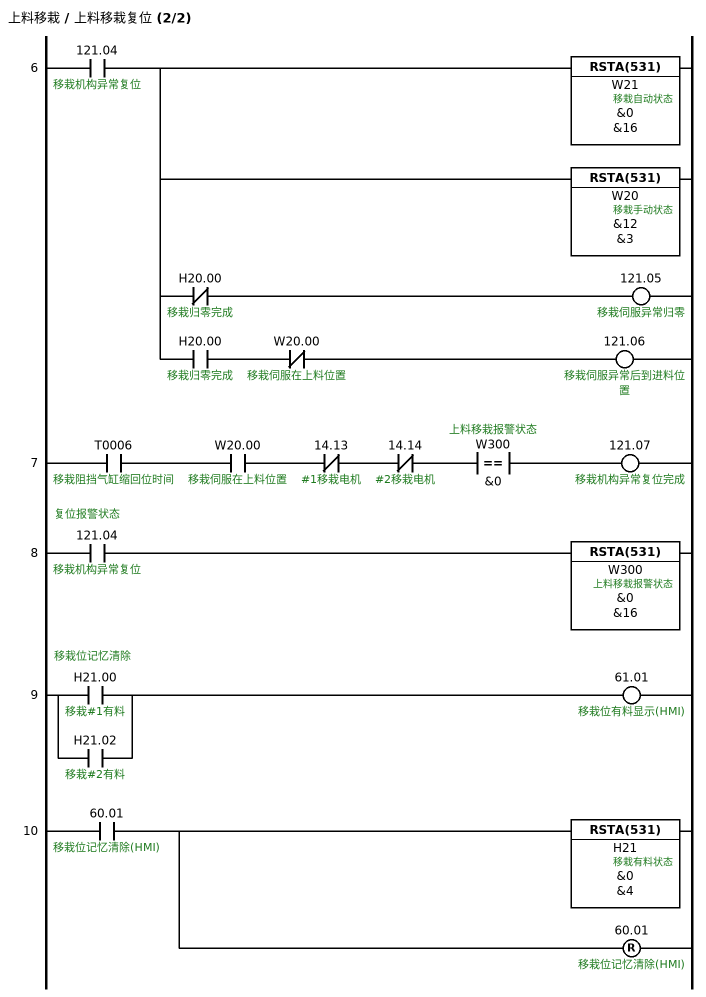
; [picture p113: 上料移栽 / 上料移栽复位, rungs 6-10]
; rung 6
LD 121.04  ; 移栽机构异常复位
OUT TR0
RSTA(531) W21 &0 &16  ; 移栽自动状态
RSTA(531) W20 &12 &3  ; 移栽手动状态
ANDNOT H20.00  ; 移栽归零完成
OUT 121.05  ; 移栽伺服异常归零
LD TR0
AND H20.00  ; 移栽归零完成
ANDNOT W20.00  ; 移栽伺服在上料位置
OUT 121.06  ; 移栽伺服异常后到进料位置
; rung 7
LD T0006  ; 移栽阻挡气缸缩回位时间
AND W20.00  ; 移栽伺服在上料位置
ANDNOT 14.13  ; #1移栽电机
ANDNOT 14.14  ; #2移栽电机
AND=(300) W300 &0  ; 上料移栽报警状态
OUT 121.07  ; 移栽机构异常复位完成
; rung 8: 复位报警状态
LD 121.04  ; 移栽机构异常复位
RSTA(531) W300 &0 &16  ; 上料移栽报警状态
; rung 9: 移栽位记忆清除
LD H21.00  ; 移栽#1有料
OR H21.02  ; 移栽#2有料
OUT 61.01  ; 移栽位有料显示(HMI)
; rung 10
LD 60.01  ; 移栽位记忆清除(HMI)
RSTA(531) H21 &0 &4  ; 移栽有料状态
RSET 60.01  ; 移栽位记忆清除(HMI)

### Section END
; rung 0
END(001)

## Program 左机械手 (cyclic task 4)

### Section 左机械手手动

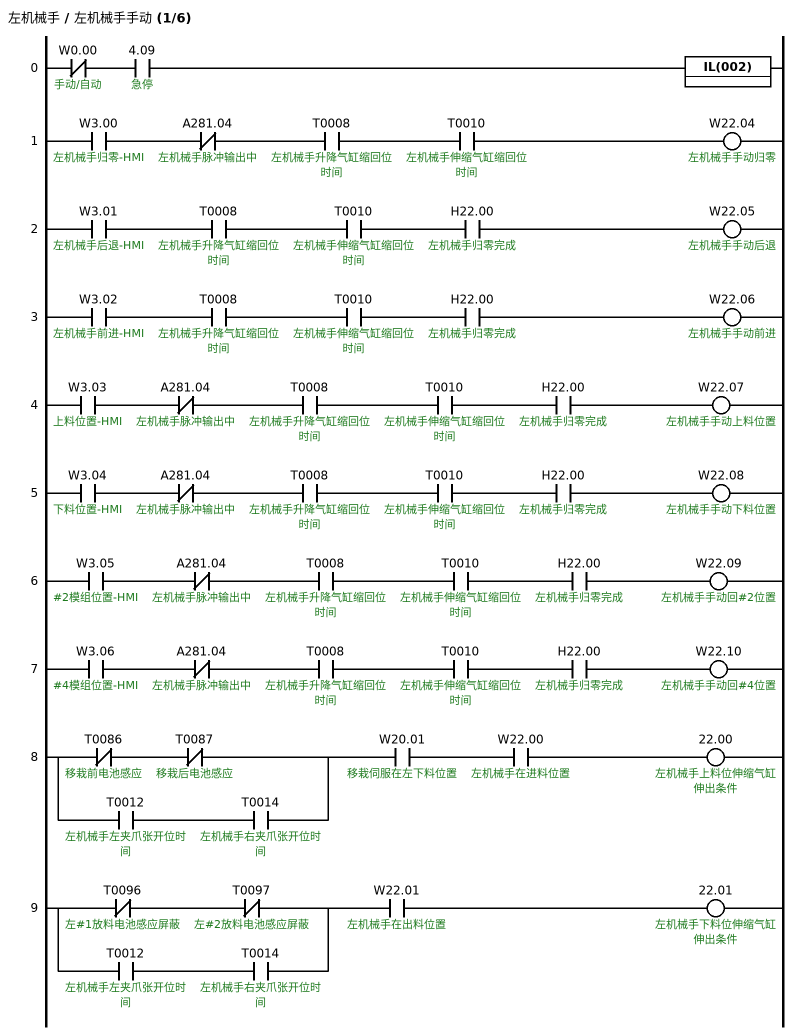
; rung 0
LDNOT W0.00  ; 手动/自动
AND 4.09  ; 急停
IL(002)
; rung 1
LD W3.00  ; 左机械手归零-HMI
ANDNOT A281.04  ; 左机械手脉冲输出中
AND T0008  ; 左机械手升降气缸缩回位时间
AND T0010  ; 左机械手伸缩气缸缩回位时间
OUT W22.04  ; 左机械手手动归零
; rung 2
LD W3.01  ; 左机械手后退-HMI
AND T0008  ; 左机械手升降气缸缩回位时间
AND T0010  ; 左机械手伸缩气缸缩回位时间
AND H22.00  ; 左机械手归零完成
OUT W22.05  ; 左机械手手动后退
; rung 3
LD W3.02  ; 左机械手前进-HMI
AND T0008  ; 左机械手升降气缸缩回位时间
AND T0010  ; 左机械手伸缩气缸缩回位时间
AND H22.00  ; 左机械手归零完成
OUT W22.06  ; 左机械手手动前进
; rung 4
LD W3.03  ; 上料位置-HMI
ANDNOT A281.04  ; 左机械手脉冲输出中
AND T0008  ; 左机械手升降气缸缩回位时间
AND T0010  ; 左机械手伸缩气缸缩回位时间
AND H22.00  ; 左机械手归零完成
OUT W22.07  ; 左机械手手动上料位置
; rung 5
LD W3.04  ; 下料位置-HMI
ANDNOT A281.04  ; 左机械手脉冲输出中
AND T0008  ; 左机械手升降气缸缩回位时间
AND T0010  ; 左机械手伸缩气缸缩回位时间
AND H22.00  ; 左机械手归零完成
OUT W22.08  ; 左机械手手动下料位置
; rung 6
LD W3.05  ; #2模组位置-HMI
ANDNOT A281.04  ; 左机械手脉冲输出中
AND T0008  ; 左机械手升降气缸缩回位时间
AND T0010  ; 左机械手伸缩气缸缩回位时间
AND H22.00  ; 左机械手归零完成
OUT W22.09  ; 左机械手手动回#2位置
; rung 7
LD W3.06  ; #4模组位置-HMI
ANDNOT A281.04  ; 左机械手脉冲输出中
AND T0008  ; 左机械手升降气缸缩回位时间
AND T0010  ; 左机械手伸缩气缸缩回位时间
AND H22.00  ; 左机械手归零完成
OUT W22.10  ; 左机械手手动回#4位置
; rung 8
LDNOT T0086  ; 移栽前电池感应
ANDNOT T0087  ; 移栽后电池感应
LD T0012  ; 左机械手左夹爪张开位时间
AND T0014  ; 左机械手右夹爪张开位时间
ORLD
AND W20.01  ; 移栽伺服在左下料位置
AND W22.00  ; 左机械手在进料位置
OUT 22.00  ; 左机械手上料位伸缩气缸伸出条件
; rung 9
LDNOT T0096  ; 左#1放料电池感应屏蔽
ANDNOT T0097  ; 左#2放料电池感应屏蔽
LD T0012  ; 左机械手左夹爪张开位时间
AND T0014  ; 左机械手右夹爪张开位时间
ORLD
AND W22.01  ; 左机械手在出料位置
OUT 22.01  ; 左机械手下料位伸缩气缸伸出条件

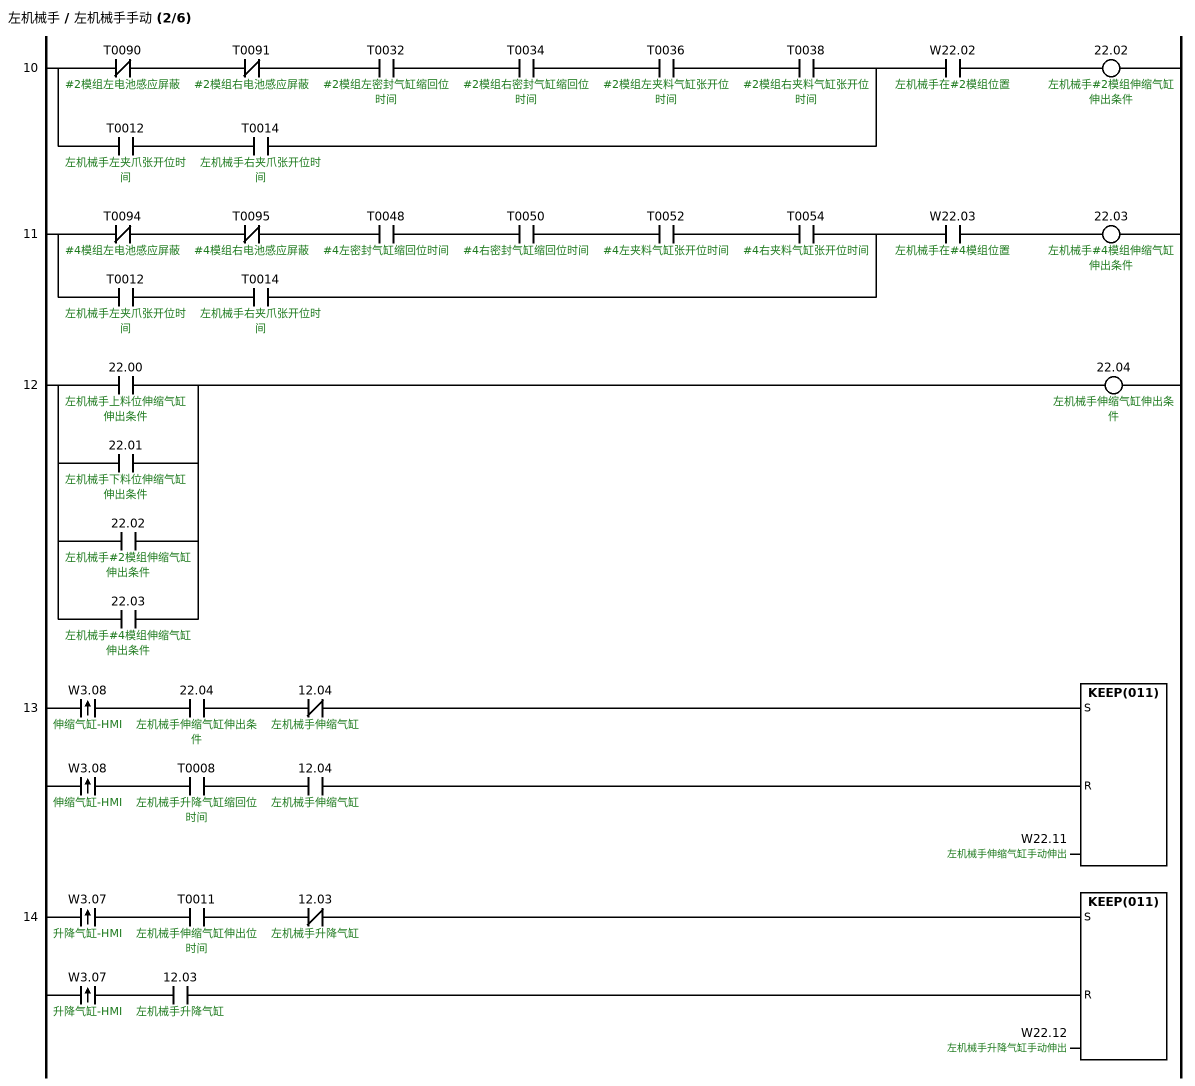
; rung 10
LDNOT T0090  ; #2模组左电池感应屏蔽
ANDNOT T0091  ; #2模组右电池感应屏蔽
AND T0032  ; #2模组左密封气缸缩回位时间
AND T0034  ; #2模组右密封气缸缩回位时间
AND T0036  ; #2模组左夹料气缸张开位时间
AND T0038  ; #2模组右夹料气缸张开位时间
LD T0012  ; 左机械手左夹爪张开位时间
AND T0014  ; 左机械手右夹爪张开位时间
ORLD
AND W22.02  ; 左机械手在#2模组位置
OUT 22.02  ; 左机械手#2模组伸缩气缸伸出条件
; rung 11
LDNOT T0094  ; #4模组左电池感应屏蔽
ANDNOT T0095  ; #4模组右电池感应屏蔽
AND T0048  ; #4左密封气缸缩回位时间
AND T0050  ; #4右密封气缸缩回位时间
AND T0052  ; #4左夹料气缸张开位时间
AND T0054  ; #4右夹料气缸张开位时间
LD T0012  ; 左机械手左夹爪张开位时间
AND T0014  ; 左机械手右夹爪张开位时间
ORLD
AND W22.03  ; 左机械手在#4模组位置
OUT 22.03  ; 左机械手#4模组伸缩气缸伸出条件
; rung 12
LD 22.00  ; 左机械手上料位伸缩气缸伸出条件
OR 22.01  ; 左机械手下料位伸缩气缸伸出条件
OR 22.02  ; 左机械手#2模组伸缩气缸伸出条件
OR 22.03  ; 左机械手#4模组伸缩气缸伸出条件
OUT 22.04  ; 左机械手伸缩气缸伸出条件
; rung 13
@LD W3.08  ; 伸缩气缸-HMI
AND 22.04  ; 左机械手伸缩气缸伸出条件
ANDNOT 12.04  ; 左机械手伸缩气缸
@LD W3.08  ; 伸缩气缸-HMI
AND T0008  ; 左机械手升降气缸缩回位时间
AND 12.04  ; 左机械手伸缩气缸
KEEP(011) W22.11  ; 左机械手伸缩气缸手动伸出
; rung 14
@LD W3.07  ; 升降气缸-HMI
AND T0011  ; 左机械手伸缩气缸伸出位时间
ANDNOT 12.03  ; 左机械手升降气缸
@LD W3.07  ; 升降气缸-HMI
AND 12.03  ; 左机械手升降气缸
KEEP(011) W22.12  ; 左机械手升降气缸手动伸出

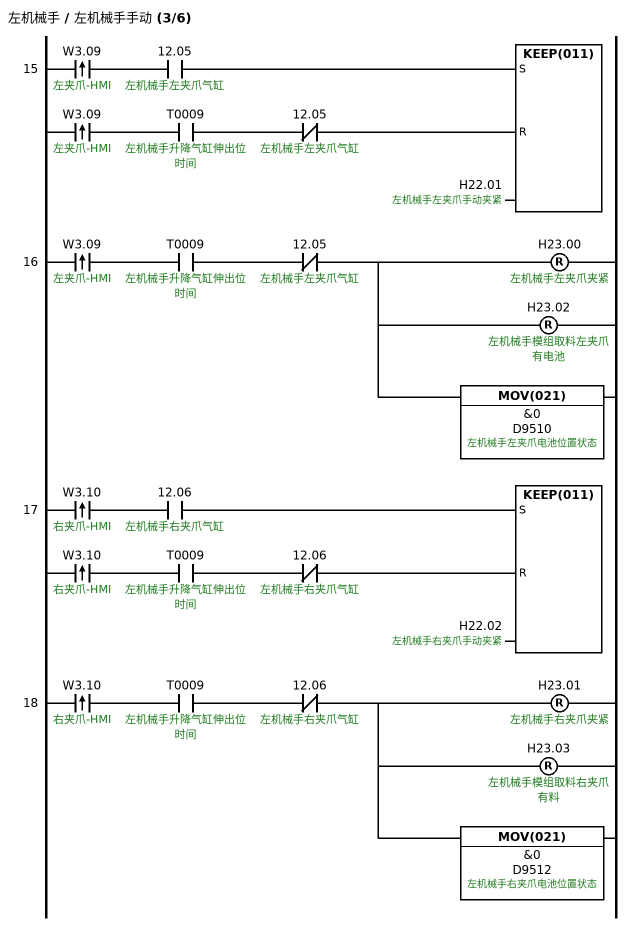
; rung 15
@LD W3.09  ; 左夹爪-HMI
AND 12.05  ; 左机械手左夹爪气缸
@LD W3.09  ; 左夹爪-HMI
AND T0009  ; 左机械手升降气缸伸出位时间
ANDNOT 12.05  ; 左机械手左夹爪气缸
KEEP(011) H22.01  ; 左机械手左夹爪手动夹紧
; rung 16
@LD W3.09  ; 左夹爪-HMI
AND T0009  ; 左机械手升降气缸伸出位时间
ANDNOT 12.05  ; 左机械手左夹爪气缸
RSET H23.00  ; 左机械手左夹爪夹紧
RSET H23.02  ; 左机械手模组取料左夹爪有电池
MOV(021) &0 D9510  ; 左机械手左夹爪电池位置状态
; rung 17
@LD W3.10  ; 右夹爪-HMI
AND 12.06  ; 左机械手右夹爪气缸
@LD W3.10  ; 右夹爪-HMI
AND T0009  ; 左机械手升降气缸伸出位时间
ANDNOT 12.06  ; 左机械手右夹爪气缸
KEEP(011) H22.02  ; 左机械手右夹爪手动夹紧
; rung 18
@LD W3.10  ; 右夹爪-HMI
AND T0009  ; 左机械手升降气缸伸出位时间
ANDNOT 12.06  ; 左机械手右夹爪气缸
RSET H23.01  ; 左机械手右夹爪夹紧
RSET H23.03  ; 左机械手模组取料右夹爪有料
MOV(021) &0 D9512  ; 左机械手右夹爪电池位置状态

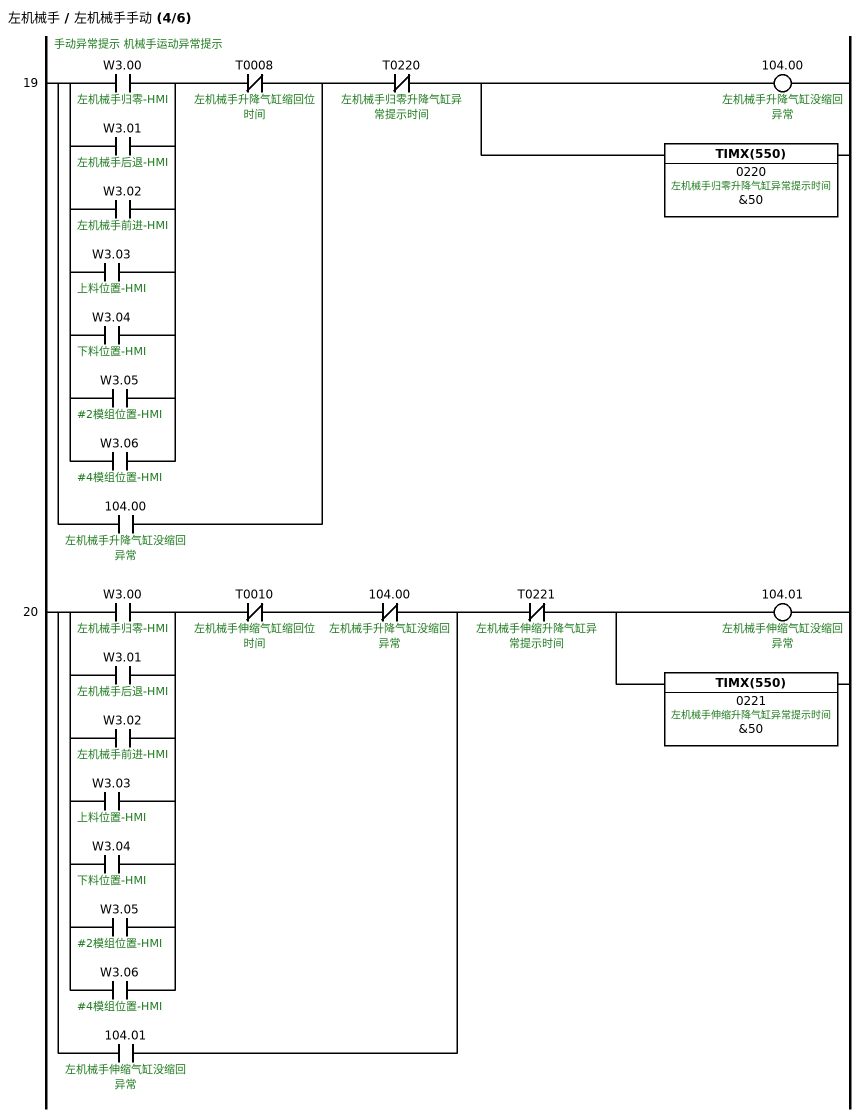
; rung 19: 手动异常提示 机械手运动异常提示
LD W3.00  ; 左机械手归零-HMI
OR W3.01  ; 左机械手后退-HMI
OR W3.02  ; 左机械手前进-HMI
OR W3.03  ; 上料位置-HMI
OR W3.04  ; 下料位置-HMI
OR W3.05  ; #2模组位置-HMI
OR W3.06  ; #4模组位置-HMI
ANDNOT T0008  ; 左机械手升降气缸缩回位时间
OR 104.00  ; 左机械手升降气缸没缩回异常
ANDNOT T0220  ; 左机械手归零升降气缸异常提示时间
OUT 104.00  ; 左机械手升降气缸没缩回异常
TIMX(550) 0220 &50  ; 左机械手归零升降气缸异常提示时间
; rung 20
LD W3.00  ; 左机械手归零-HMI
OR W3.01  ; 左机械手后退-HMI
OR W3.02  ; 左机械手前进-HMI
OR W3.03  ; 上料位置-HMI
OR W3.04  ; 下料位置-HMI
OR W3.05  ; #2模组位置-HMI
OR W3.06  ; #4模组位置-HMI
ANDNOT T0010  ; 左机械手伸缩气缸缩回位时间
ANDNOT 104.00  ; 左机械手升降气缸没缩回异常
OR 104.01  ; 左机械手伸缩气缸没缩回异常
ANDNOT T0221  ; 左机械手伸缩升降气缸异常提示时间
OUT 104.01  ; 左机械手伸缩气缸没缩回异常
TIMX(550) 0221 &50  ; 左机械手伸缩升降气缸异常提示时间

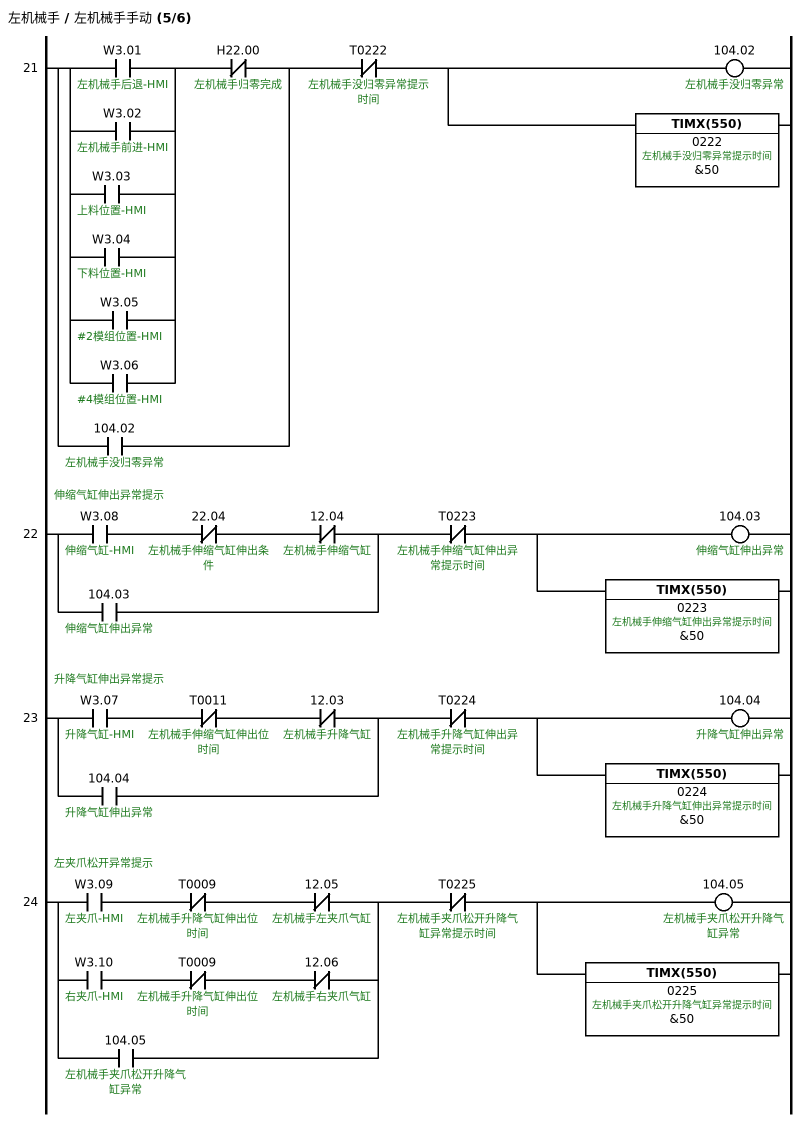
; rung 21
LD W3.01  ; 左机械手后退-HMI
OR W3.02  ; 左机械手前进-HMI
OR W3.03  ; 上料位置-HMI
OR W3.04  ; 下料位置-HMI
OR W3.05  ; #2模组位置-HMI
OR W3.06  ; #4模组位置-HMI
ANDNOT H22.00  ; 左机械手归零完成
OR 104.02  ; 左机械手没归零异常
ANDNOT T0222  ; 左机械手没归零异常提示时间
OUT 104.02  ; 左机械手没归零异常
TIMX(550) 0222 &50  ; 左机械手没归零异常提示时间
; rung 22: 伸缩气缸伸出异常提示
LD W3.08  ; 伸缩气缸-HMI
ANDNOT 22.04  ; 左机械手伸缩气缸伸出条件
ANDNOT 12.04  ; 左机械手伸缩气缸
OR 104.03  ; 伸缩气缸伸出异常
ANDNOT T0223  ; 左机械手伸缩气缸伸出异常提示时间
OUT 104.03  ; 伸缩气缸伸出异常
TIMX(550) 0223 &50  ; 左机械手伸缩气缸伸出异常提示时间
; rung 23: 升降气缸伸出异常提示
LD W3.07  ; 升降气缸-HMI
ANDNOT T0011  ; 左机械手伸缩气缸伸出位时间
ANDNOT 12.03  ; 左机械手升降气缸
OR 104.04  ; 升降气缸伸出异常
ANDNOT T0224  ; 左机械手升降气缸伸出异常提示时间
OUT 104.04  ; 升降气缸伸出异常
TIMX(550) 0224 &50  ; 左机械手升降气缸伸出异常提示时间
; rung 24: 左夹爪松开异常提示
LD W3.09  ; 左夹爪-HMI
ANDNOT T0009  ; 左机械手升降气缸伸出位时间
ANDNOT 12.05  ; 左机械手左夹爪气缸
LD W3.10  ; 右夹爪-HMI
ANDNOT T0009  ; 左机械手升降气缸伸出位时间
ANDNOT 12.06  ; 左机械手右夹爪气缸
ORLD
OR 104.05  ; 左机械手夹爪松开升降气缸异常
ANDNOT T0225  ; 左机械手夹爪松开升降气缸异常提示时间
OUT 104.05  ; 左机械手夹爪松开升降气缸异常
TIMX(550) 0225 &50  ; 左机械手夹爪松开升降气缸异常提示时间

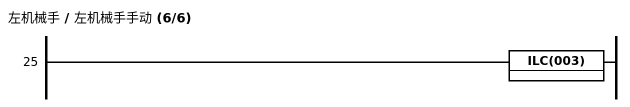
; rung 25
ILC(003)

### Section 左机械手自动

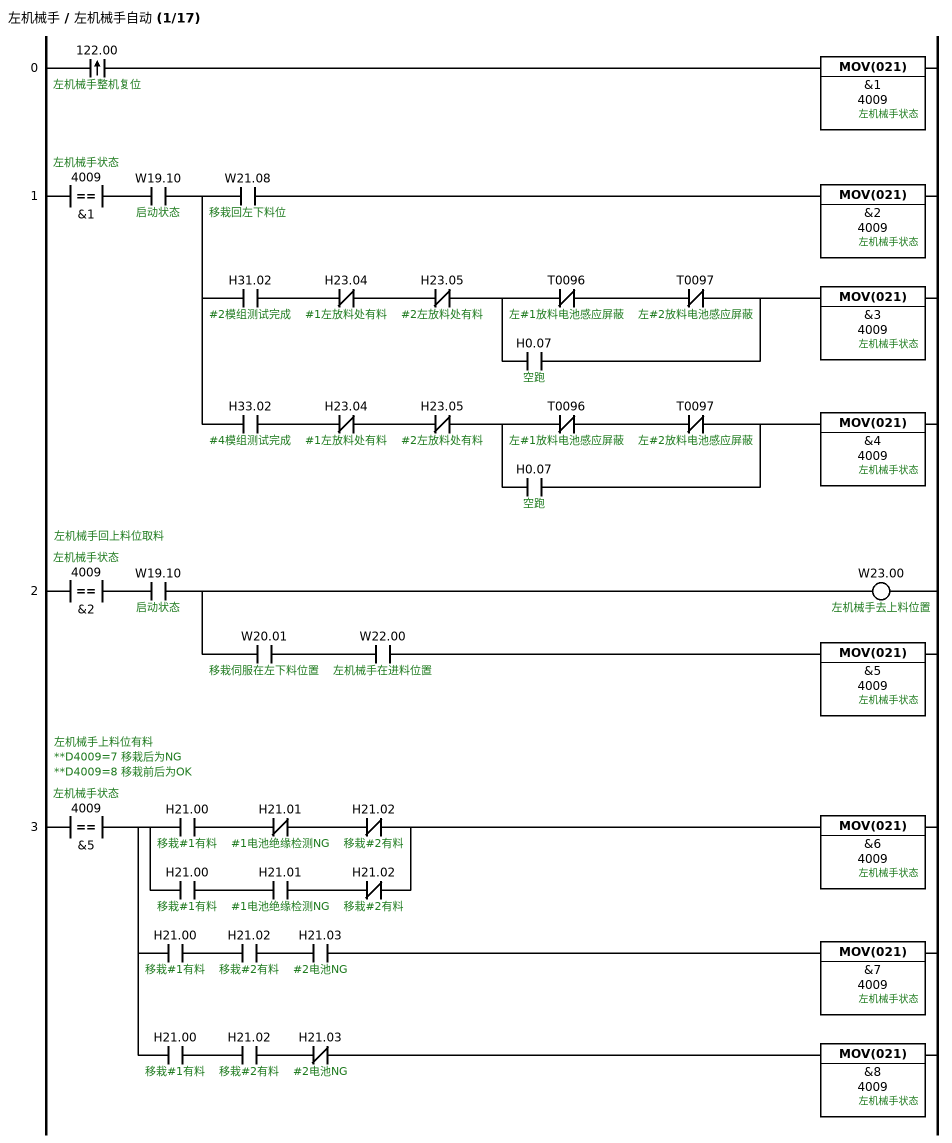
; rung 0
@LD 122.00  ; 左机械手整机复位
MOV(021) &1 4009  ; 左机械手状态
; rung 1
LD=(300) 4009 &1  ; 左机械手状态
AND W19.10  ; 启动状态
OUT TR0
AND W21.08  ; 移栽回左下料位
MOV(021) &2 4009  ; 左机械手状态
LD TR0
AND H31.02  ; #2模组测试完成
ANDNOT H23.04  ; #1左放料处有料
ANDNOT H23.05  ; #2左放料处有料
LDNOT T0096  ; 左#1放料电池感应屏蔽
ANDNOT T0097  ; 左#2放料电池感应屏蔽
OR H0.07  ; 空跑
ANDLD
MOV(021) &3 4009  ; 左机械手状态
LD TR0
AND H33.02  ; #4模组测试完成
ANDNOT H23.04  ; #1左放料处有料
ANDNOT H23.05  ; #2左放料处有料
LDNOT T0096  ; 左#1放料电池感应屏蔽
ANDNOT T0097  ; 左#2放料电池感应屏蔽
OR H0.07  ; 空跑
ANDLD
MOV(021) &4 4009  ; 左机械手状态
; rung 2: 左机械手回上料位取料
LD=(300) 4009 &2  ; 左机械手状态
AND W19.10  ; 启动状态
OUT W23.00  ; 左机械手去上料位置
AND W20.01  ; 移栽伺服在左下料位置
AND W22.00  ; 左机械手在进料位置
MOV(021) &5 4009  ; 左机械手状态
; rung 3: 左机械手上料位有料 / **D4009=7 移栽后为NG / **D4009=8 移栽前后为OK
LD=(300) 4009 &5  ; 左机械手状态
OUT TR0
LD H21.00  ; 移栽#1有料
ANDNOT H21.01  ; #1电池绝缘检测NG
ANDNOT H21.02  ; 移栽#2有料
LD H21.00  ; 移栽#1有料
AND H21.01  ; #1电池绝缘检测NG
ANDNOT H21.02  ; 移栽#2有料
ORLD
ANDLD
MOV(021) &6 4009  ; 左机械手状态
LD TR0
AND H21.00  ; 移栽#1有料
AND H21.02  ; 移栽#2有料
AND H21.03  ; #2电池NG
MOV(021) &7 4009  ; 左机械手状态
LD TR0
AND H21.00  ; 移栽#1有料
AND H21.02  ; 移栽#2有料
ANDNOT H21.03  ; #2电池NG
MOV(021) &8 4009  ; 左机械手状态

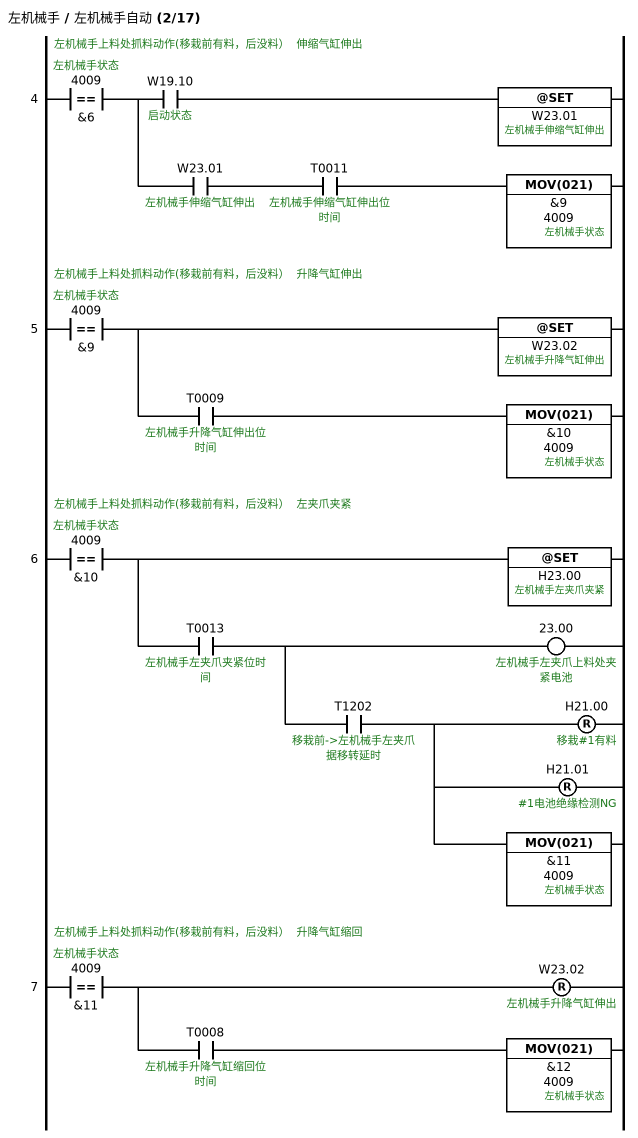
; rung 4: 左机械手上料处抓料动作(移栽前有料，后没料）  伸缩气缸伸出
LD=(300) 4009 &6  ; 左机械手状态
OUT TR0
AND W19.10  ; 启动状态
@SET W23.01  ; 左机械手伸缩气缸伸出
LD TR0
AND W23.01  ; 左机械手伸缩气缸伸出
AND T0011  ; 左机械手伸缩气缸伸出位时间
MOV(021) &9 4009  ; 左机械手状态
; rung 5: 左机械手上料处抓料动作(移栽前有料，后没料）  升降气缸伸出
LD=(300) 4009 &9  ; 左机械手状态
@SET W23.02  ; 左机械手升降气缸伸出
AND T0009  ; 左机械手升降气缸伸出位时间
MOV(021) &10 4009  ; 左机械手状态
; rung 6: 左机械手上料处抓料动作(移栽前有料，后没料）  左夹爪夹紧
LD=(300) 4009 &10  ; 左机械手状态
@SET H23.00  ; 左机械手左夹爪夹紧
AND T0013  ; 左机械手左夹爪夹紧位时间
OUT 23.00  ; 左机械手左夹爪上料处夹紧电池
AND T1202  ; 移栽前->左机械手左夹爪据移转延时
RSET H21.00  ; 移栽#1有料
RSET H21.01  ; #1电池绝缘检测NG
MOV(021) &11 4009  ; 左机械手状态
; rung 7: 左机械手上料处抓料动作(移栽前有料，后没料）  升降气缸缩回
LD=(300) 4009 &11  ; 左机械手状态
RSET W23.02  ; 左机械手升降气缸伸出
AND T0008  ; 左机械手升降气缸缩回位时间
MOV(021) &12 4009  ; 左机械手状态

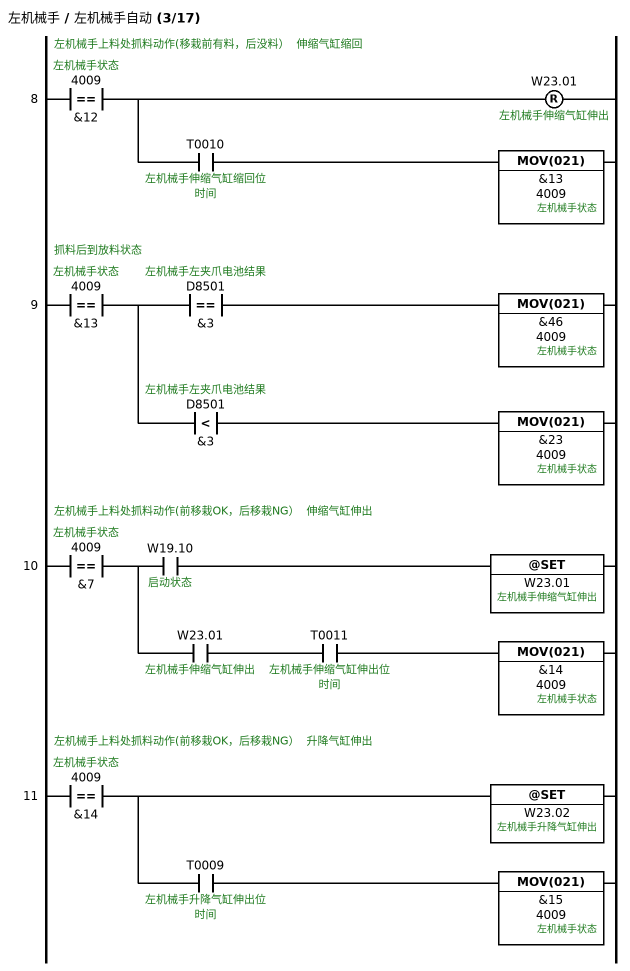
; rung 8: 左机械手上料处抓料动作(移栽前有料，后没料）  伸缩气缸缩回
LD=(300) 4009 &12  ; 左机械手状态
RSET W23.01  ; 左机械手伸缩气缸伸出
AND T0010  ; 左机械手伸缩气缸缩回位时间
MOV(021) &13 4009  ; 左机械手状态
; rung 9: 抓料后到放料状态
LD=(300) 4009 &13  ; 左机械手状态
OUT TR0
AND=(300) D8501 &3  ; 左机械手左夹爪电池结果
MOV(021) &46 4009  ; 左机械手状态
LD TR0
AND<(310) D8501 &3  ; 左机械手左夹爪电池结果
MOV(021) &23 4009  ; 左机械手状态
; rung 10: 左机械手上料处抓料动作(前移栽OK，后移栽NG）  伸缩气缸伸出
LD=(300) 4009 &7  ; 左机械手状态
OUT TR0
AND W19.10  ; 启动状态
@SET W23.01  ; 左机械手伸缩气缸伸出
LD TR0
AND W23.01  ; 左机械手伸缩气缸伸出
AND T0011  ; 左机械手伸缩气缸伸出位时间
MOV(021) &14 4009  ; 左机械手状态
; rung 11: 左机械手上料处抓料动作(前移栽OK，后移栽NG）  升降气缸伸出
LD=(300) 4009 &14  ; 左机械手状态
@SET W23.02  ; 左机械手升降气缸伸出
AND T0009  ; 左机械手升降气缸伸出位时间
MOV(021) &15 4009  ; 左机械手状态

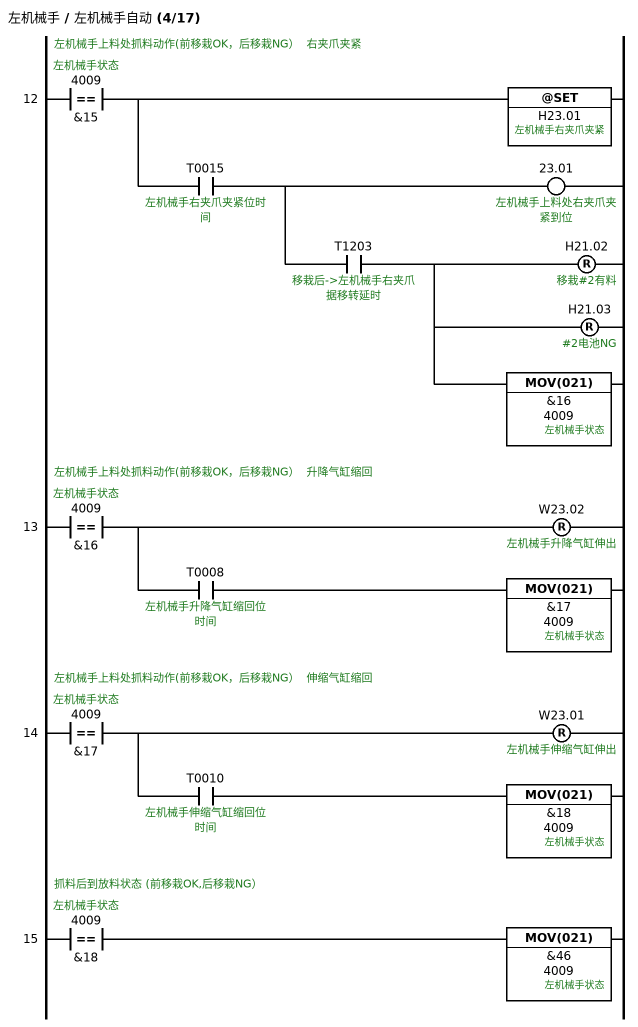
; rung 12: 左机械手上料处抓料动作(前移栽OK，后移栽NG）  右夹爪夹紧
LD=(300) 4009 &15  ; 左机械手状态
@SET H23.01  ; 左机械手右夹爪夹紧
AND T0015  ; 左机械手右夹爪夹紧位时间
OUT 23.01  ; 左机械手上料处右夹爪夹紧到位
AND T1203  ; 移栽后->左机械手右夹爪据移转延时
RSET H21.02  ; 移栽#2有料
RSET H21.03  ; #2电池NG
MOV(021) &16 4009  ; 左机械手状态
; rung 13: 左机械手上料处抓料动作(前移栽OK，后移栽NG）  升降气缸缩回
LD=(300) 4009 &16  ; 左机械手状态
RSET W23.02  ; 左机械手升降气缸伸出
AND T0008  ; 左机械手升降气缸缩回位时间
MOV(021) &17 4009  ; 左机械手状态
; rung 14: 左机械手上料处抓料动作(前移栽OK，后移栽NG）  伸缩气缸缩回
LD=(300) 4009 &17  ; 左机械手状态
RSET W23.01  ; 左机械手伸缩气缸伸出
AND T0010  ; 左机械手伸缩气缸缩回位时间
MOV(021) &18 4009  ; 左机械手状态
; rung 15: 抓料后到放料状态 (前移栽OK,后移栽NG）
LD=(300) 4009 &18  ; 左机械手状态
MOV(021) &46 4009  ; 左机械手状态

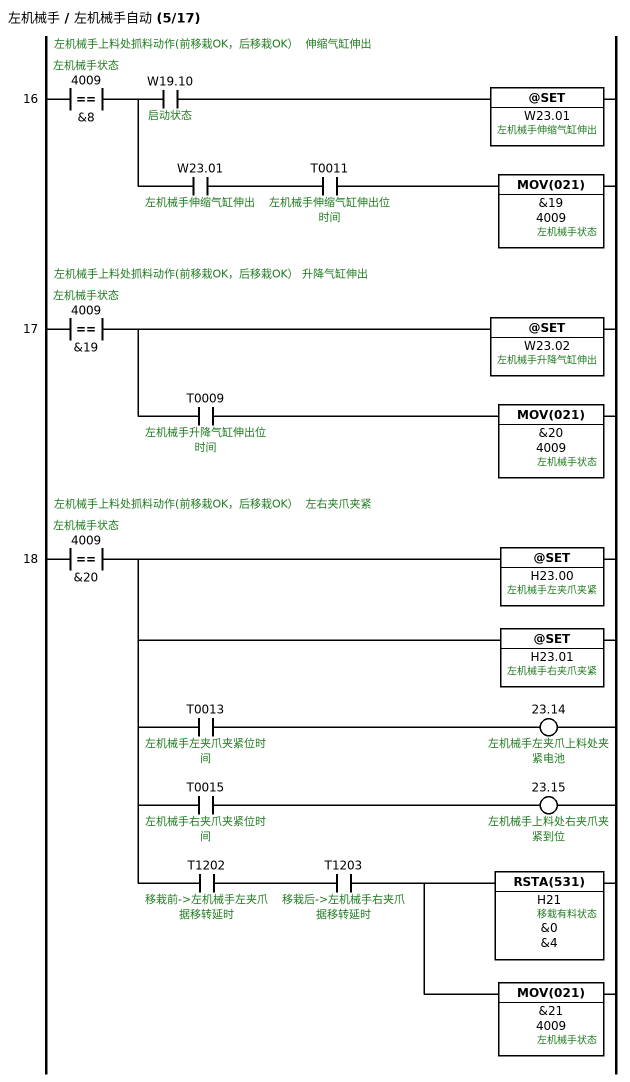
; rung 16: 左机械手上料处抓料动作(前移栽OK，后移栽OK）  伸缩气缸伸出
LD=(300) 4009 &8  ; 左机械手状态
OUT TR0
AND W19.10  ; 启动状态
@SET W23.01  ; 左机械手伸缩气缸伸出
LD TR0
AND W23.01  ; 左机械手伸缩气缸伸出
AND T0011  ; 左机械手伸缩气缸伸出位时间
MOV(021) &19 4009  ; 左机械手状态
; rung 17: 左机械手上料处抓料动作(前移栽OK，后移栽OK） 升降气缸伸出
LD=(300) 4009 &19  ; 左机械手状态
@SET W23.02  ; 左机械手升降气缸伸出
AND T0009  ; 左机械手升降气缸伸出位时间
MOV(021) &20 4009  ; 左机械手状态
; rung 18: 左机械手上料处抓料动作(前移栽OK，后移栽OK）  左右夹爪夹紧
LD=(300) 4009 &20  ; 左机械手状态
OUT TR0
@SET H23.00  ; 左机械手左夹爪夹紧
@SET H23.01  ; 左机械手右夹爪夹紧
AND T0013  ; 左机械手左夹爪夹紧位时间
OUT 23.14  ; 左机械手左夹爪上料处夹紧电池
LD TR0
AND T0015  ; 左机械手右夹爪夹紧位时间
OUT 23.15  ; 左机械手上料处右夹爪夹紧到位
LD TR0
AND T1202  ; 移栽前->左机械手左夹爪据移转延时
AND T1203  ; 移栽后->左机械手右夹爪据移转延时
RSTA(531) H21 &0 &4  ; 移栽有料状态
MOV(021) &21 4009  ; 左机械手状态

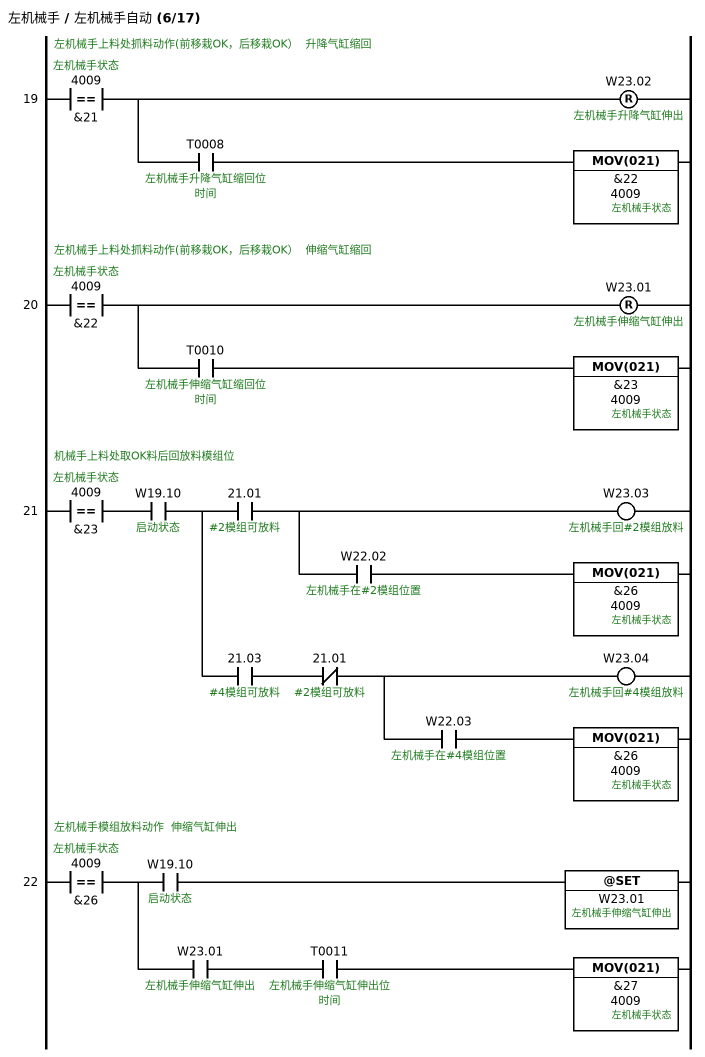
; rung 19: 左机械手上料处抓料动作(前移栽OK，后移栽OK）  升降气缸缩回
LD=(300) 4009 &21  ; 左机械手状态
RSET W23.02  ; 左机械手升降气缸伸出
AND T0008  ; 左机械手升降气缸缩回位时间
MOV(021) &22 4009  ; 左机械手状态
; rung 20: 左机械手上料处抓料动作(前移栽OK，后移栽OK）  伸缩气缸缩回
LD=(300) 4009 &22  ; 左机械手状态
RSET W23.01  ; 左机械手伸缩气缸伸出
AND T0010  ; 左机械手伸缩气缸缩回位时间
MOV(021) &23 4009  ; 左机械手状态
; rung 21: 机械手上料处取OK料后回放料模组位
LD=(300) 4009 &23  ; 左机械手状态
AND W19.10  ; 启动状态
OUT TR0
AND 21.01  ; #2模组可放料
OUT W23.03  ; 左机械手回#2模组放料
AND W22.02  ; 左机械手在#2模组位置
MOV(021) &26 4009  ; 左机械手状态
LD TR0
AND 21.03  ; #4模组可放料
ANDNOT 21.01  ; #2模组可放料
OUT W23.04  ; 左机械手回#4模组放料
AND W22.03  ; 左机械手在#4模组位置
MOV(021) &26 4009  ; 左机械手状态
; rung 22: 左机械手模组放料动作  伸缩气缸伸出
LD=(300) 4009 &26  ; 左机械手状态
OUT TR0
AND W19.10  ; 启动状态
@SET W23.01  ; 左机械手伸缩气缸伸出
LD TR0
AND W23.01  ; 左机械手伸缩气缸伸出
AND T0011  ; 左机械手伸缩气缸伸出位时间
MOV(021) &27 4009  ; 左机械手状态

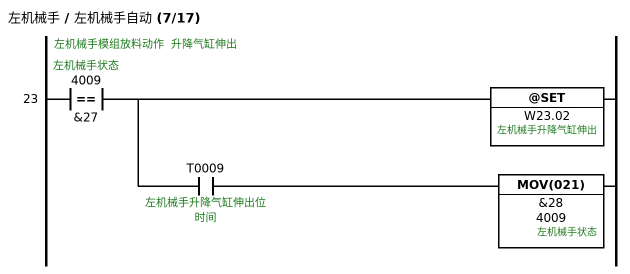
; rung 23: 左机械手模组放料动作  升降气缸伸出
LD=(300) 4009 &27  ; 左机械手状态
@SET W23.02  ; 左机械手升降气缸伸出
AND T0009  ; 左机械手升降气缸伸出位时间
MOV(021) &28 4009  ; 左机械手状态

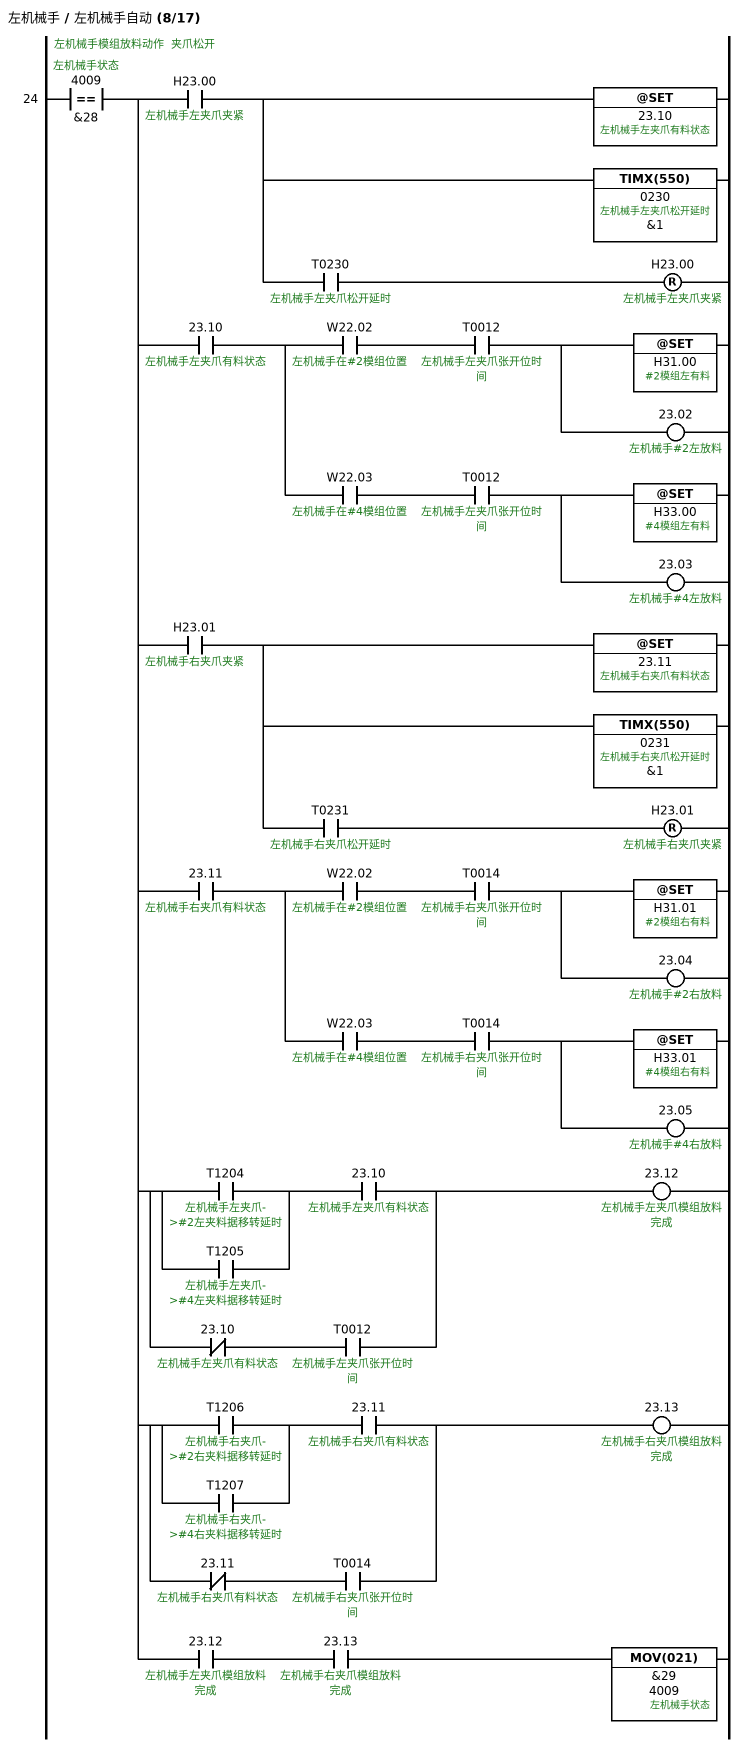
; rung 24: 左机械手模组放料动作  夹爪松开
LD=(300) 4009 &28  ; 左机械手状态
OUT TR0
AND H23.00  ; 左机械手左夹爪夹紧
@SET 23.10  ; 左机械手左夹爪有料状态
TIMX(550) 0230 &1  ; 左机械手左夹爪松开延时
AND T0230  ; 左机械手左夹爪松开延时
RSET H23.00  ; 左机械手左夹爪夹紧
LD TR0
AND 23.10  ; 左机械手左夹爪有料状态
OUT TR1
AND W22.02  ; 左机械手在#2模组位置
AND T0012  ; 左机械手左夹爪张开位时间
@SET H31.00  ; #2模组左有料
OUT 23.02  ; 左机械手#2左放料
LD TR1
AND W22.03  ; 左机械手在#4模组位置
AND T0012  ; 左机械手左夹爪张开位时间
@SET H33.00  ; #4模组左有料
OUT 23.03  ; 左机械手#4左放料
LD TR0
AND H23.01  ; 左机械手右夹爪夹紧
@SET 23.11  ; 左机械手右夹爪有料状态
TIMX(550) 0231 &1  ; 左机械手右夹爪松开延时
AND T0231  ; 左机械手右夹爪松开延时
RSET H23.01  ; 左机械手右夹爪夹紧
LD TR0
AND 23.11  ; 左机械手右夹爪有料状态
OUT TR1
AND W22.02  ; 左机械手在#2模组位置
AND T0014  ; 左机械手右夹爪张开位时间
@SET H31.01  ; #2模组右有料
OUT 23.04  ; 左机械手#2右放料
LD TR1
AND W22.03  ; 左机械手在#4模组位置
AND T0014  ; 左机械手右夹爪张开位时间
@SET H33.01  ; #4模组右有料
OUT 23.05  ; 左机械手#4右放料
LD TR0
LD T1204  ; 左机械手左夹爪->#2左夹料据移转延时
OR T1205  ; 左机械手左夹爪->#4左夹料据移转延时
AND 23.10  ; 左机械手左夹爪有料状态
LDNOT 23.10  ; 左机械手左夹爪有料状态
AND T0012  ; 左机械手左夹爪张开位时间
ORLD
ANDLD
OUT 23.12  ; 左机械手左夹爪模组放料完成
LD TR0
LD T1206  ; 左机械手右夹爪->#2右夹料据移转延时
OR T1207  ; 左机械手右夹爪->#4右夹料据移转延时
AND 23.11  ; 左机械手右夹爪有料状态
LDNOT 23.11  ; 左机械手右夹爪有料状态
AND T0014  ; 左机械手右夹爪张开位时间
ORLD
ANDLD
OUT 23.13  ; 左机械手右夹爪模组放料完成
LD TR0
AND 23.12  ; 左机械手左夹爪模组放料完成
AND 23.13  ; 左机械手右夹爪模组放料完成
MOV(021) &29 4009  ; 左机械手状态

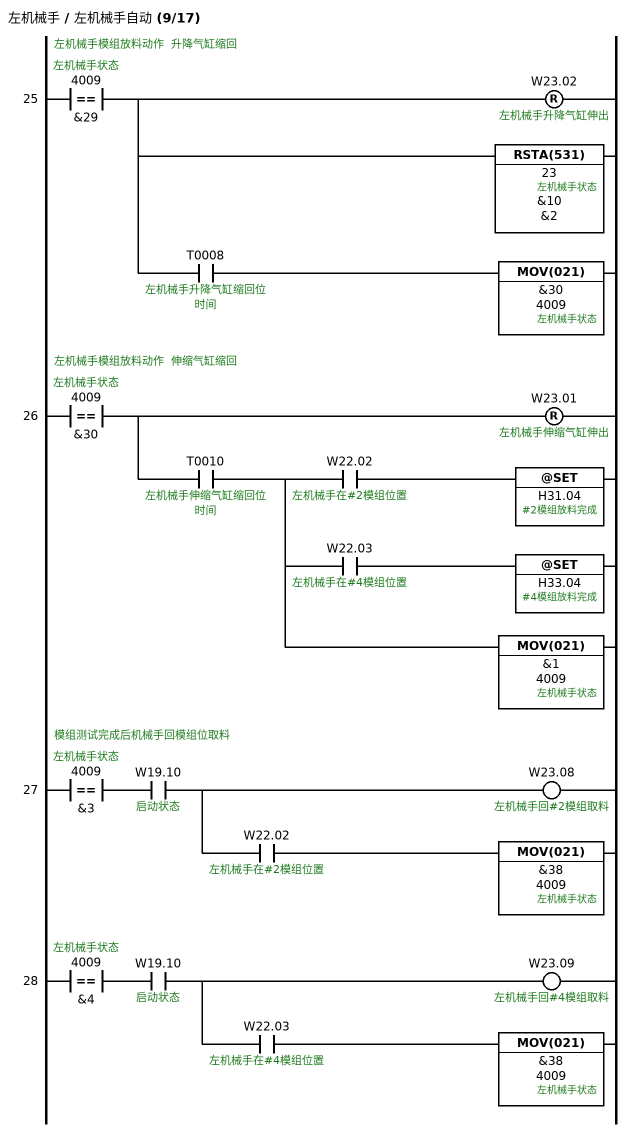
; rung 25: 左机械手模组放料动作  升降气缸缩回
LD=(300) 4009 &29  ; 左机械手状态
RSET W23.02  ; 左机械手升降气缸伸出
RSTA(531) 23 &10 &2  ; 左机械手状态
AND T0008  ; 左机械手升降气缸缩回位时间
MOV(021) &30 4009  ; 左机械手状态
; rung 26: 左机械手模组放料动作  伸缩气缸缩回
LD=(300) 4009 &30  ; 左机械手状态
RSET W23.01  ; 左机械手伸缩气缸伸出
AND T0010  ; 左机械手伸缩气缸缩回位时间
OUT TR0
AND W22.02  ; 左机械手在#2模组位置
@SET H31.04  ; #2模组放料完成
LD TR0
AND W22.03  ; 左机械手在#4模组位置
@SET H33.04  ; #4模组放料完成
LD TR0
MOV(021) &1 4009  ; 左机械手状态
; rung 27: 模组测试完成后机械手回模组位取料
LD=(300) 4009 &3  ; 左机械手状态
AND W19.10  ; 启动状态
OUT W23.08  ; 左机械手回#2模组取料
AND W22.02  ; 左机械手在#2模组位置
MOV(021) &38 4009  ; 左机械手状态
; rung 28
LD=(300) 4009 &4  ; 左机械手状态
AND W19.10  ; 启动状态
OUT W23.09  ; 左机械手回#4模组取料
AND W22.03  ; 左机械手在#4模组位置
MOV(021) &38 4009  ; 左机械手状态

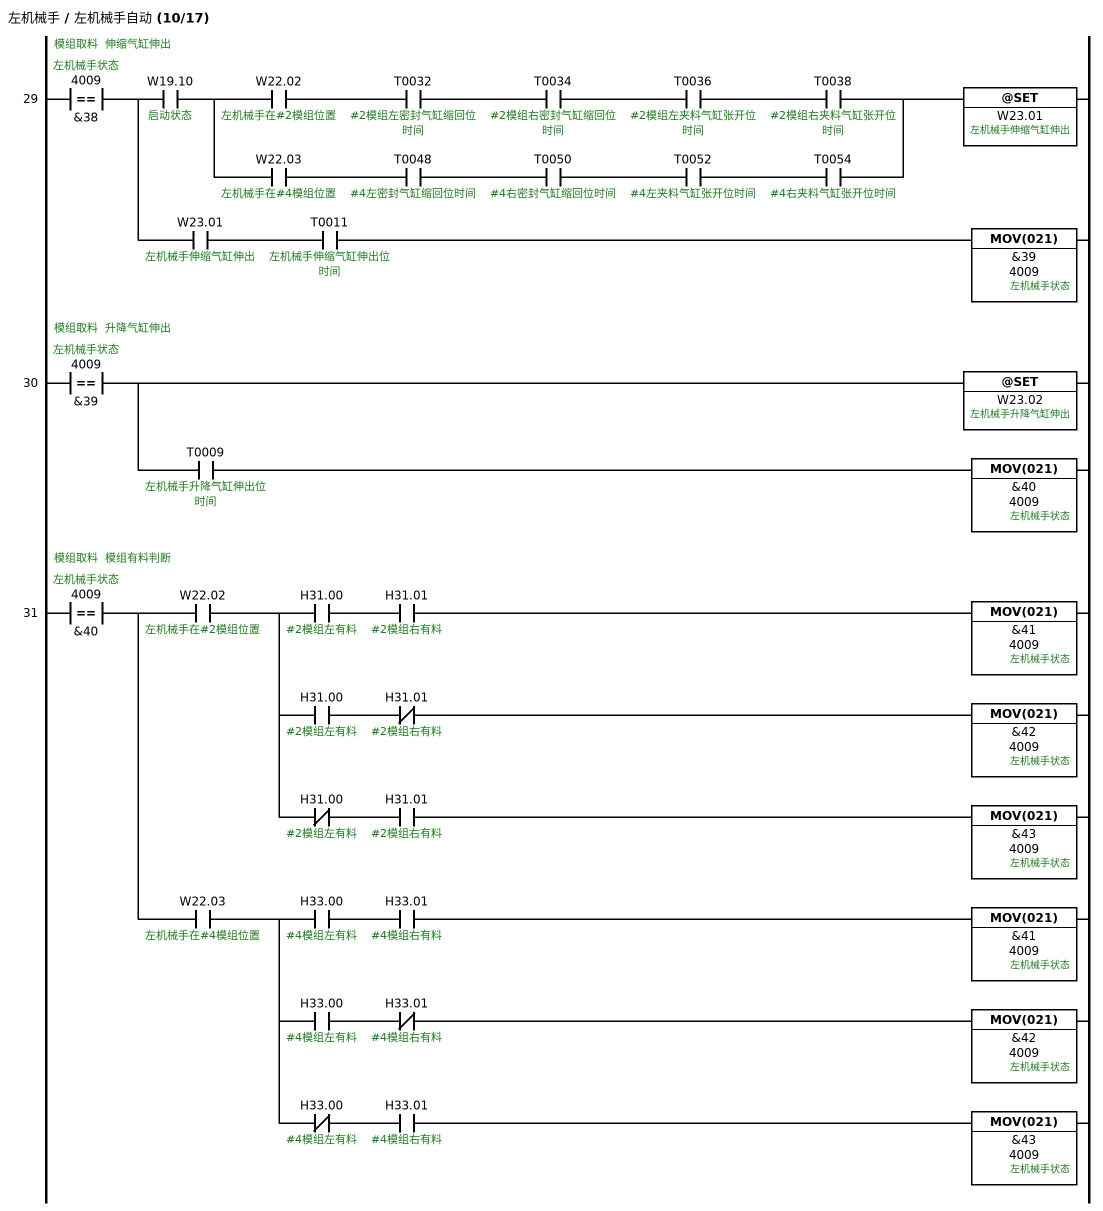
; rung 29: 模组取料  伸缩气缸伸出
LD=(300) 4009 &38  ; 左机械手状态
OUT TR0
AND W19.10  ; 启动状态
LD W22.02  ; 左机械手在#2模组位置
AND T0032  ; #2模组左密封气缸缩回位时间
AND T0034  ; #2模组右密封气缸缩回位时间
AND T0036  ; #2模组左夹料气缸张开位时间
AND T0038  ; #2模组右夹料气缸张开位时间
LD W22.03  ; 左机械手在#4模组位置
AND T0048  ; #4左密封气缸缩回位时间
AND T0050  ; #4右密封气缸缩回位时间
AND T0052  ; #4左夹料气缸张开位时间
AND T0054  ; #4右夹料气缸张开位时间
ORLD
ANDLD
@SET W23.01  ; 左机械手伸缩气缸伸出
LD TR0
AND W23.01  ; 左机械手伸缩气缸伸出
AND T0011  ; 左机械手伸缩气缸伸出位时间
MOV(021) &39 4009  ; 左机械手状态
; rung 30: 模组取料  升降气缸伸出
LD=(300) 4009 &39  ; 左机械手状态
@SET W23.02  ; 左机械手升降气缸伸出
AND T0009  ; 左机械手升降气缸伸出位时间
MOV(021) &40 4009  ; 左机械手状态
; rung 31: 模组取料  模组有料判断
LD=(300) 4009 &40  ; 左机械手状态
OUT TR0
AND W22.02  ; 左机械手在#2模组位置
OUT TR1
AND H31.00  ; #2模组左有料
AND H31.01  ; #2模组右有料
MOV(021) &41 4009  ; 左机械手状态
LD TR1
AND H31.00  ; #2模组左有料
ANDNOT H31.01  ; #2模组右有料
MOV(021) &42 4009  ; 左机械手状态
LD TR1
ANDNOT H31.00  ; #2模组左有料
AND H31.01  ; #2模组右有料
MOV(021) &43 4009  ; 左机械手状态
LD TR0
AND W22.03  ; 左机械手在#4模组位置
OUT TR0
AND H33.00  ; #4模组左有料
AND H33.01  ; #4模组右有料
MOV(021) &41 4009  ; 左机械手状态
LD TR0
AND H33.00  ; #4模组左有料
ANDNOT H33.01  ; #4模组右有料
MOV(021) &42 4009  ; 左机械手状态
LD TR0
ANDNOT H33.00  ; #4模组左有料
AND H33.01  ; #4模组右有料
MOV(021) &43 4009  ; 左机械手状态

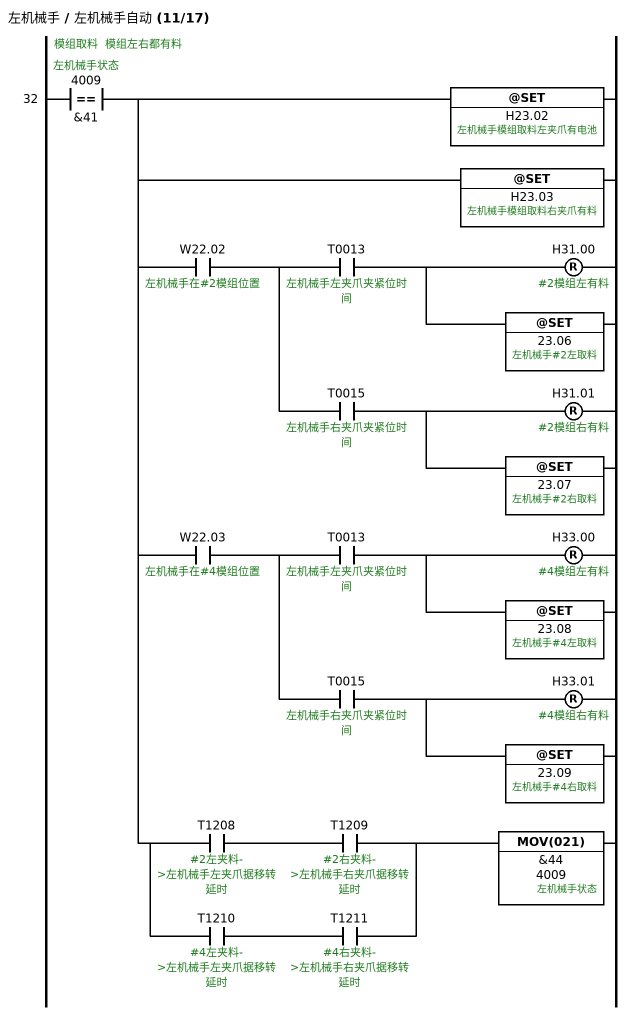
; rung 32: 模组取料  模组左右都有料
LD=(300) 4009 &41  ; 左机械手状态
OUT TR0
@SET H23.02  ; 左机械手模组取料左夹爪有电池
@SET H23.03  ; 左机械手模组取料右夹爪有料
AND W22.02  ; 左机械手在#2模组位置
OUT TR1
AND T0013  ; 左机械手左夹爪夹紧位时间
RSET H31.00  ; #2模组左有料
@SET 23.06  ; 左机械手#2左取料
LD TR1
AND T0015  ; 左机械手右夹爪夹紧位时间
RSET H31.01  ; #2模组右有料
@SET 23.07  ; 左机械手#2右取料
LD TR0
AND W22.03  ; 左机械手在#4模组位置
OUT TR1
AND T0013  ; 左机械手左夹爪夹紧位时间
RSET H33.00  ; #4模组左有料
@SET 23.08  ; 左机械手#4左取料
LD TR1
AND T0015  ; 左机械手右夹爪夹紧位时间
RSET H33.01  ; #4模组右有料
@SET 23.09  ; 左机械手#4右取料
LD TR0
LD T1208  ; #2左夹料->左机械手左夹爪据移转延时
AND T1209  ; #2右夹料->左机械手右夹爪据移转延时
LD T1210  ; #4左夹料->左机械手左夹爪据移转延时
AND T1211  ; #4右夹料->左机械手右夹爪据移转延时
ORLD
ANDLD
MOV(021) &44 4009  ; 左机械手状态

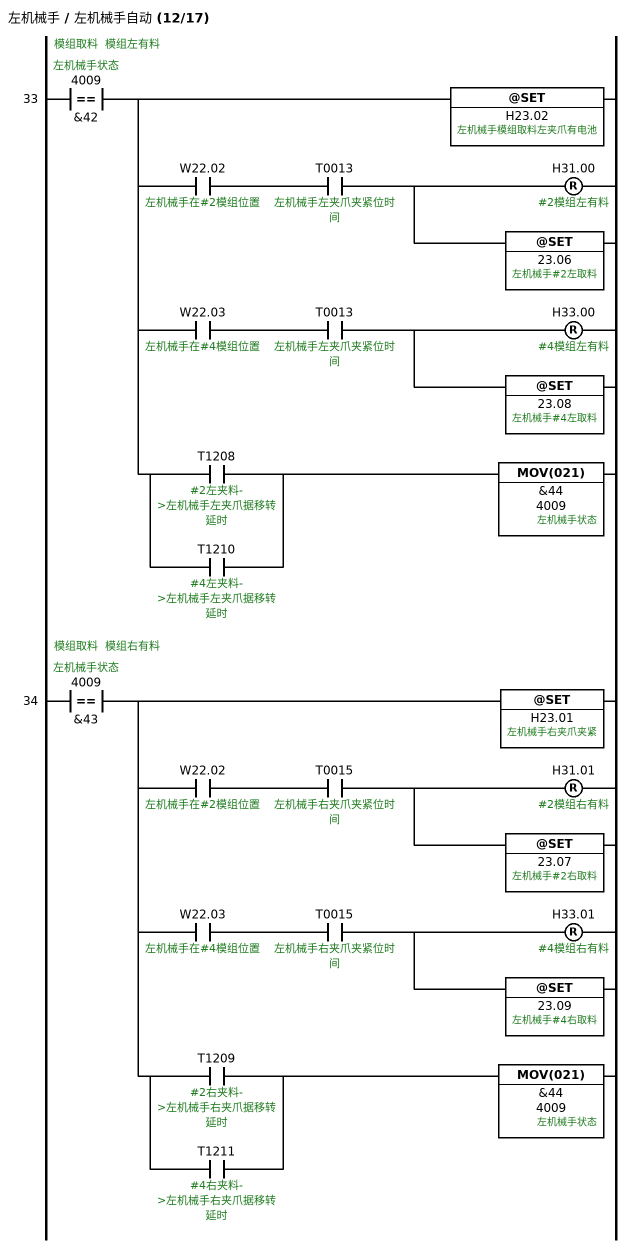
; rung 33: 模组取料  模组左有料
LD=(300) 4009 &42  ; 左机械手状态
OUT TR0
@SET H23.02  ; 左机械手模组取料左夹爪有电池
AND W22.02  ; 左机械手在#2模组位置
AND T0013  ; 左机械手左夹爪夹紧位时间
RSET H31.00  ; #2模组左有料
@SET 23.06  ; 左机械手#2左取料
LD TR0
AND W22.03  ; 左机械手在#4模组位置
AND T0013  ; 左机械手左夹爪夹紧位时间
RSET H33.00  ; #4模组左有料
@SET 23.08  ; 左机械手#4左取料
LD TR0
LD T1208  ; #2左夹料->左机械手左夹爪据移转延时
OR T1210  ; #4左夹料->左机械手左夹爪据移转延时
ANDLD
MOV(021) &44 4009  ; 左机械手状态
; rung 34: 模组取料  模组右有料
LD=(300) 4009 &43  ; 左机械手状态
OUT TR0
@SET H23.01  ; 左机械手右夹爪夹紧
AND W22.02  ; 左机械手在#2模组位置
AND T0015  ; 左机械手右夹爪夹紧位时间
RSET H31.01  ; #2模组右有料
@SET 23.07  ; 左机械手#2右取料
LD TR0
AND W22.03  ; 左机械手在#4模组位置
AND T0015  ; 左机械手右夹爪夹紧位时间
RSET H33.01  ; #4模组右有料
@SET 23.09  ; 左机械手#4右取料
LD TR0
LD T1209  ; #2右夹料->左机械手右夹爪据移转延时
OR T1211  ; #4右夹料->左机械手右夹爪据移转延时
ANDLD
MOV(021) &44 4009  ; 左机械手状态

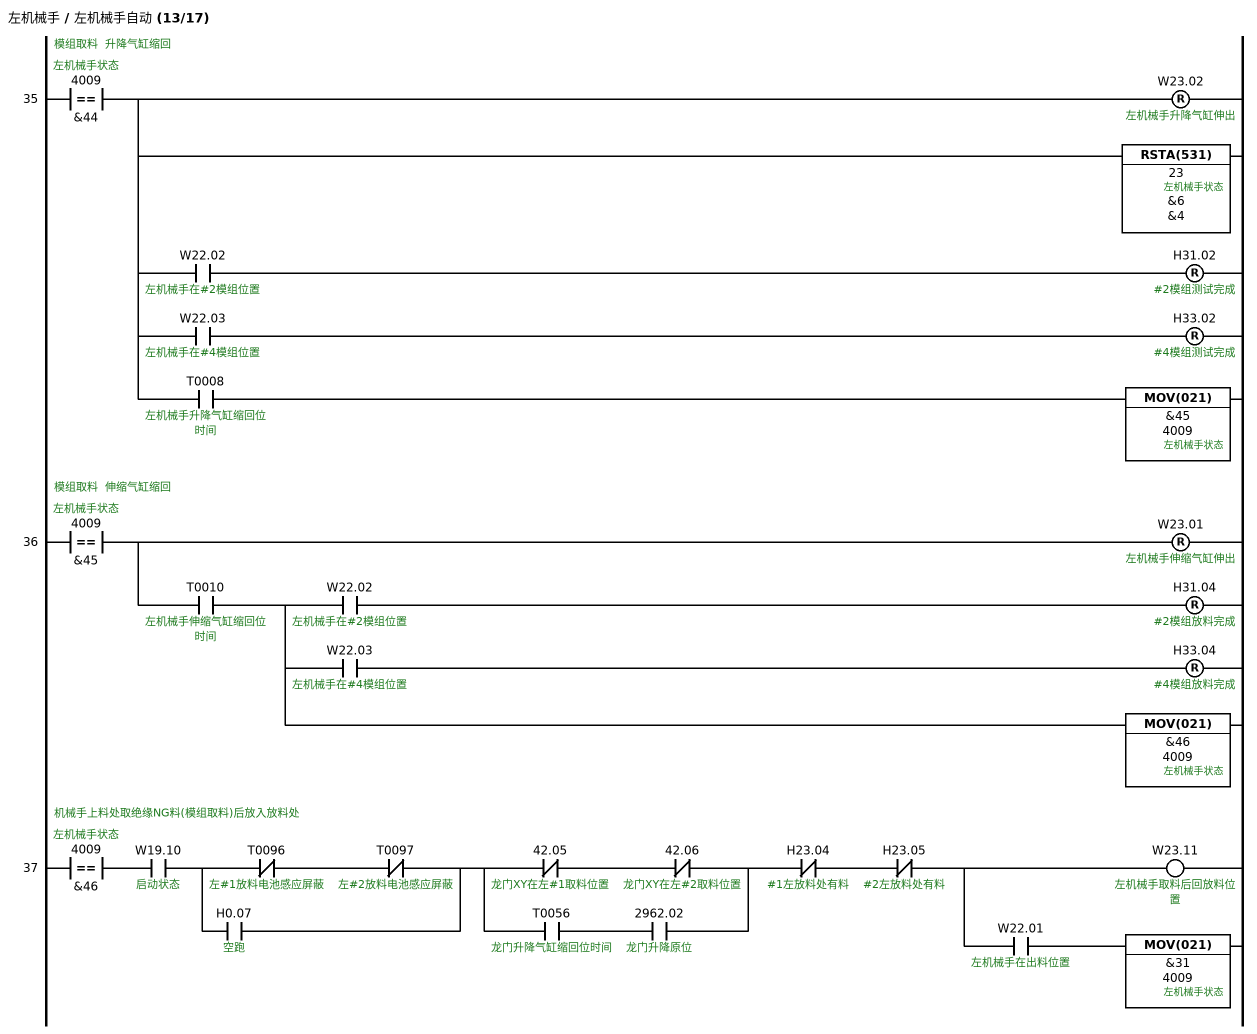
; rung 35: 模组取料  升降气缸缩回
LD=(300) 4009 &44  ; 左机械手状态
OUT TR0
RSET W23.02  ; 左机械手升降气缸伸出
RSTA(531) 23 &6 &4  ; 左机械手状态
AND W22.02  ; 左机械手在#2模组位置
RSET H31.02  ; #2模组测试完成
LD TR0
AND W22.03  ; 左机械手在#4模组位置
RSET H33.02  ; #4模组测试完成
LD TR0
AND T0008  ; 左机械手升降气缸缩回位时间
MOV(021) &45 4009  ; 左机械手状态
; rung 36: 模组取料  伸缩气缸缩回
LD=(300) 4009 &45  ; 左机械手状态
RSET W23.01  ; 左机械手伸缩气缸伸出
AND T0010  ; 左机械手伸缩气缸缩回位时间
OUT TR0
AND W22.02  ; 左机械手在#2模组位置
RSET H31.04  ; #2模组放料完成
LD TR0
AND W22.03  ; 左机械手在#4模组位置
RSET H33.04  ; #4模组放料完成
LD TR0
MOV(021) &46 4009  ; 左机械手状态
; rung 37: 机械手上料处取绝缘NG料(模组取料)后放入放料处
LD=(300) 4009 &46  ; 左机械手状态
AND W19.10  ; 启动状态
LDNOT T0096  ; 左#1放料电池感应屏蔽
ANDNOT T0097  ; 左#2放料电池感应屏蔽
OR H0.07  ; 空跑
ANDLD
LDNOT 42.05  ; 龙门XY在左#1取料位置
ANDNOT 42.06  ; 龙门XY在左#2取料位置
LD T0056  ; 龙门升降气缸缩回位时间
AND 2962.02  ; 龙门升降原位
ORLD
ANDLD
ANDNOT H23.04  ; #1左放料处有料
ANDNOT H23.05  ; #2左放料处有料
OUT W23.11  ; 左机械手取料后回放料位置
AND W22.01  ; 左机械手在出料位置
MOV(021) &31 4009  ; 左机械手状态

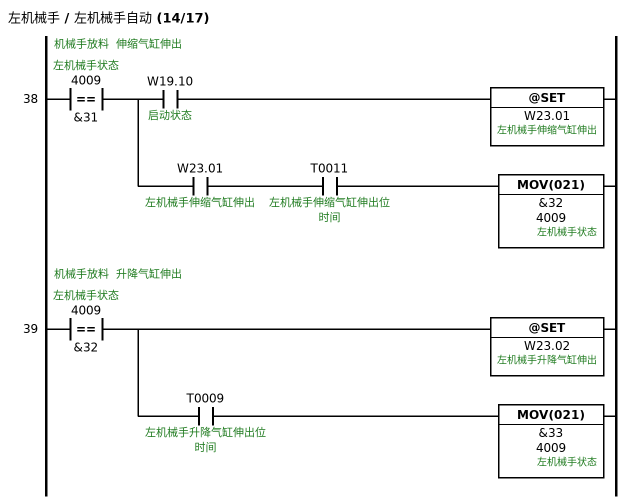
; rung 38: 机械手放料  伸缩气缸伸出
LD=(300) 4009 &31  ; 左机械手状态
OUT TR0
AND W19.10  ; 启动状态
@SET W23.01  ; 左机械手伸缩气缸伸出
LD TR0
AND W23.01  ; 左机械手伸缩气缸伸出
AND T0011  ; 左机械手伸缩气缸伸出位时间
MOV(021) &32 4009  ; 左机械手状态
; rung 39: 机械手放料  升降气缸伸出
LD=(300) 4009 &32  ; 左机械手状态
@SET W23.02  ; 左机械手升降气缸伸出
AND T0009  ; 左机械手升降气缸伸出位时间
MOV(021) &33 4009  ; 左机械手状态

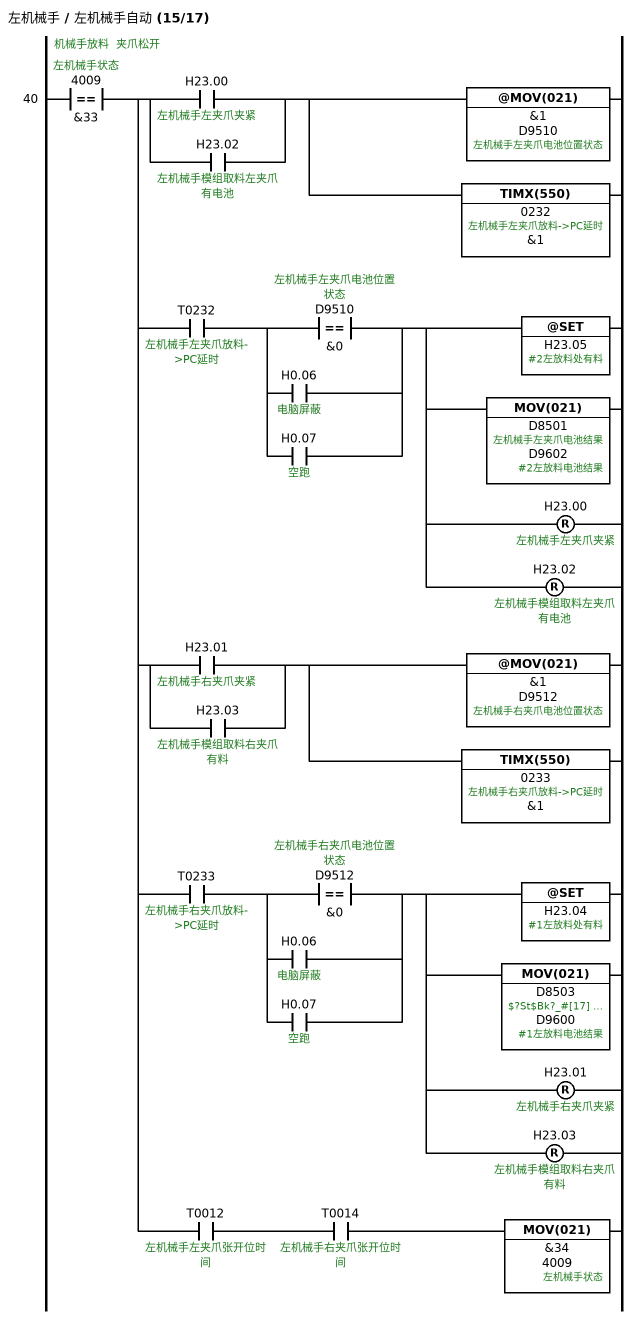
; rung 40: 机械手放料  夹爪松开
LD=(300) 4009 &33  ; 左机械手状态
OUT TR0
LD H23.00  ; 左机械手左夹爪夹紧
OR H23.02  ; 左机械手模组取料左夹爪有电池
ANDLD
@MOV(021) &1 D9510  ; 左机械手左夹爪电池位置状态
TIMX(550) 0232 &1  ; 左机械手左夹爪放料->PC延时
LD TR0
AND T0232  ; 左机械手左夹爪放料->PC延时
LD=(300) D9510 &0  ; 左机械手左夹爪电池位置状态
OR H0.06  ; 电脑屏蔽
OR H0.07  ; 空跑
ANDLD
@SET H23.05  ; #2左放料处有料
MOV(021) D8501 D9602  ; 左机械手左夹爪电池结果, #2左放料电池结果
RSET H23.00  ; 左机械手左夹爪夹紧
RSET H23.02  ; 左机械手模组取料左夹爪有电池
LD TR0
LD H23.01  ; 左机械手右夹爪夹紧
OR H23.03  ; 左机械手模组取料右夹爪有料
ANDLD
@MOV(021) &1 D9512  ; 左机械手右夹爪电池位置状态
TIMX(550) 0233 &1  ; 左机械手右夹爪放料->PC延时
LD TR0
AND T0233  ; 左机械手右夹爪放料->PC延时
LD=(300) D9512 &0  ; 左机械手右夹爪电池位置状态
OR H0.06  ; 电脑屏蔽
OR H0.07  ; 空跑
ANDLD
@SET H23.04  ; #1左放料处有料
MOV(021) D8503 D9600  ; $?St$Bk?_#[17] / 左机械手右夹爪电池结果$?St$Bk?_#[17], #1左放料电池结果
RSET H23.01  ; 左机械手右夹爪夹紧
RSET H23.03  ; 左机械手模组取料右夹爪有料
LD TR0
AND T0012  ; 左机械手左夹爪张开位时间
AND T0014  ; 左机械手右夹爪张开位时间
MOV(021) &34 4009  ; 左机械手状态

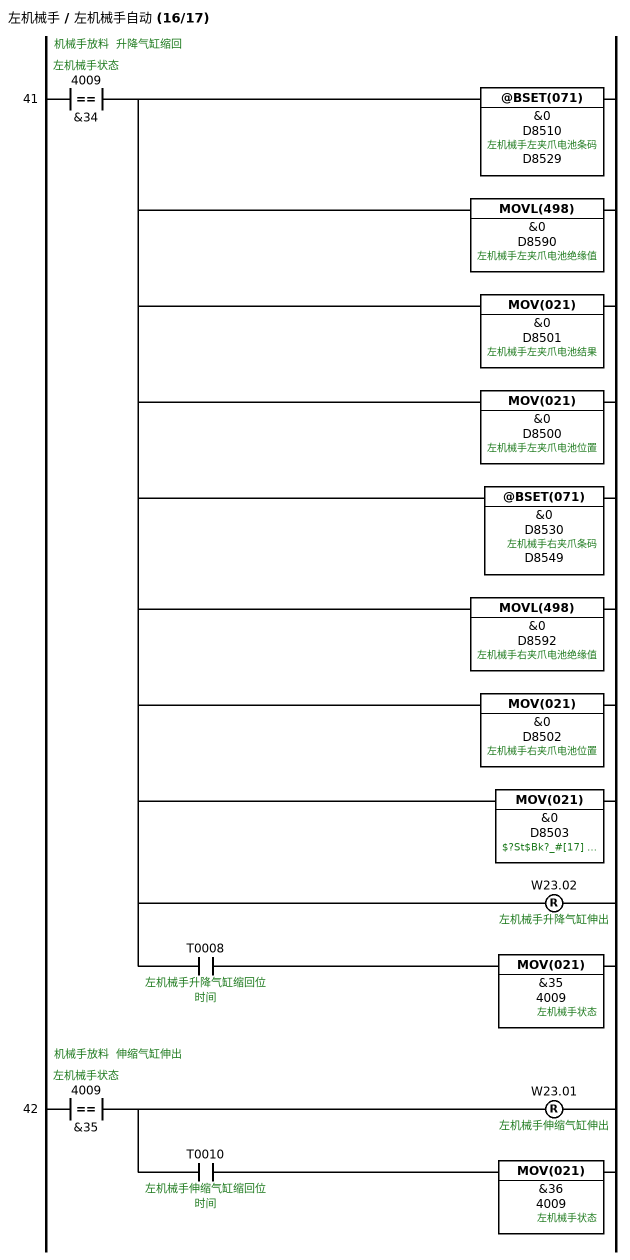
; rung 41: 机械手放料  升降气缸缩回
LD=(300) 4009 &34  ; 左机械手状态
@BSET(071) &0 D8510 D8529  ; 左机械手左夹爪电池条码
MOVL(498) &0 D8590  ; 左机械手左夹爪电池绝缘值
MOV(021) &0 D8501  ; 左机械手左夹爪电池结果
MOV(021) &0 D8500  ; 左机械手左夹爪电池位置
@BSET(071) &0 D8530 D8549  ; 左机械手右夹爪条码
MOVL(498) &0 D8592  ; 左机械手右夹爪电池绝缘值
MOV(021) &0 D8502  ; 左机械手右夹爪电池位置
MOV(021) &0 D8503  ; $?St$Bk?_#[17] / 左机械手右夹爪电池结果$?St$Bk?_#[17]
RSET W23.02  ; 左机械手升降气缸伸出
AND T0008  ; 左机械手升降气缸缩回位时间
MOV(021) &35 4009  ; 左机械手状态
; rung 42: 机械手放料  伸缩气缸伸出
LD=(300) 4009 &35  ; 左机械手状态
RSET W23.01  ; 左机械手伸缩气缸伸出
AND T0010  ; 左机械手伸缩气缸缩回位时间
MOV(021) &36 4009  ; 左机械手状态

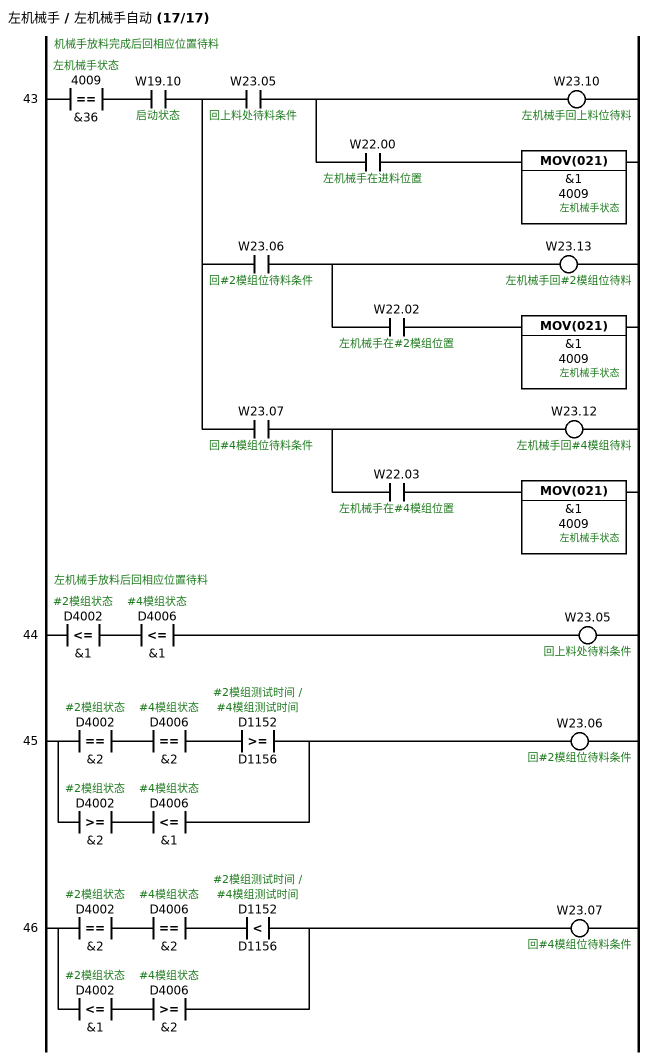
; rung 43: 机械手放料完成后回相应位置待料
LD=(300) 4009 &36  ; 左机械手状态
AND W19.10  ; 启动状态
OUT TR0
AND W23.05  ; 回上料处待料条件
OUT W23.10  ; 左机械手回上料位待料
AND W22.00  ; 左机械手在进料位置
MOV(021) &1 4009  ; 左机械手状态
LD TR0
AND W23.06  ; 回#2模组位待料条件
OUT W23.13  ; 左机械手回#2模组位待料
AND W22.02  ; 左机械手在#2模组位置
MOV(021) &1 4009  ; 左机械手状态
LD TR0
AND W23.07  ; 回#4模组位待料条件
OUT W23.12  ; 左机械手回#4模组待料
AND W22.03  ; 左机械手在#4模组位置
MOV(021) &1 4009  ; 左机械手状态
; rung 44: 左机械手放料后回相应位置待料
LD<=(315) D4002 &1  ; #2模组状态
AND<=(315) D4006 &1  ; #4模组状态
OUT W23.05  ; 回上料处待料条件
; rung 45
LD=(300) D4002 &2  ; #2模组状态
AND=(300) D4006 &2  ; #4模组状态
AND>=(325) D1152 D1156  ; #2模组测试时间, #4模组测试时间
LD>=(325) D4002 &2  ; #2模组状态
AND<=(315) D4006 &1  ; #4模组状态
ORLD
OUT W23.06  ; 回#2模组位待料条件
; rung 46
LD=(300) D4002 &2  ; #2模组状态
AND=(300) D4006 &2  ; #4模组状态
AND<(310) D1152 D1156  ; #2模组测试时间, #4模组测试时间
LD<=(315) D4002 &1  ; #2模组状态
AND>=(325) D4006 &2  ; #4模组状态
ORLD
OUT W23.07  ; 回#4模组位待料条件

### Section 伺服参数

